// TwinCAT 3 PLC project PLC
// ProgramVersion: 3.1.4024.0
// libraries:
//   SPT Base Types, * (Beckhoff Automation LLC)
//   SPT Components, * (Beckhoff Automation LLC)
//   SPT Diagnostic, * (Beckhoff Automation LLC)
//   SPT EtherCat, * (Beckhoff Automation LLC)
//   SPT Event Logger, * (Beckhoff Automation LLC)
//   SPT Kinematics, * (Beckhoff Automation LLC)
//   SPT Motion Control, * (Beckhoff Automation LLC)
//   SPT NCI, * (Beckhoff Automation LLC)
//   SPT Utilities, * (Beckhoff Automation LLC)
//   SPT Vision, * (Beckhoff Automation LLC)
//   SPT XTS, * (Beckhoff Automation LLC)
//   Tc2_MC2_Camming, * (Beckhoff Automation GmbH)
//   Tc2_Standard, * (Beckhoff Automation GmbH)
//   Tc2_System, * (Beckhoff Automation GmbH)
//   Tc3_Module, * (Beckhoff Automation GmbH)
//   VisuDialogs, * (System)
//   Tc2_EtherCAT,newest,Beckhoff Automation GmbH
//   Tc2_Math,newest,Beckhoff Automation GmbH
//   Tc2_MC2,newest,Beckhoff Automation GmbH
//   Tc2_MC2_Drive,newest,Beckhoff Automation GmbH
//   Tc2_Utilities,newest,Beckhoff Automation GmbH
//   Tc3_EventLogger,newest,Beckhoff Automation GmbH
//   Tc3_IPCDiag,newest,Beckhoff Automation GmbH
//   Tc3_JsonXml,newest,Beckhoff Automation GmbH
//   Tc3_MC2_AdvancedHoming,newest,Beckhoff Automation GmbH
//   Tc3_PackML_V2,newest,Beckhoff Automation GmbH
// project tree:
//   / GlobalTextList.TcGTLO (not stored), PlcTask.TcTTO (not stored), Visualization Manager.TcVMO (not stored)
//   Machine/EquipmentModules/ FB_MainDrive.TcPOU, FB_Station1.TcPOU, FB_Station2.TcPOU, FB_Station3.TcPOU, FB_Station4.TcPOU, FB_Station5.TcPOU
//   Machine/MachineModule/ FB_Machine.TcPOU
//   POUs/ MAIN.TcPOU
//   VISUs/ V_Operation.TcVIS, V_Machine.TcVIS
// real-time tasks:
//   TASK PlcTask: cycle T#10ms, priority 20, ADS port 350
// motion (NC):
//   TASK NC-Task 1 SAF: cycle T#2ms, priority 4, ADS port 501
//   TASK NC-Task 1 SVB: cycle T#10ms, priority 8, ADS port 511
//   AXIS Fixed Axis (id 2)
//   AXIS Variable Axis (id 3)
//   AXIS Virtual Cammed Axis (id 4)
//   AXIS Cammed Axis (id 5)
//   AXIS Virtual Offset Master Axis 4 (id 8)
//   AXIS Offset Axis (id 7)
//   AXIS Virtual Cammed Master Axis (id 9)
//   AXIS Cammed Offset Axis (id 10)
//   AXIS Virtual Offset Master Axis 5 (id 6)
//   AXIS Machine Virtual Axis (id 1)
// variable links:
//   PLC/PLC Instance <-> NC-Task 1 SAF/Axes/Cammed Axis
//     PlcTask Inputs/MAIN.Machine.Station3.CammedAxis.BasicSlaveAxis._Axis.NcToPlc <-> Outputs/ToPlc
//     PlcTask Outputs/MAIN.Machine.Station3.CammedAxis.BasicSlaveAxis._Axis.PlcToNc <-> Inputs/FromPlc
//   PLC/PLC Instance <-> NC-Task 1 SAF/Axes/Cammed Offset Axis
//     PlcTask Inputs/MAIN.Machine.Station5.CammedOffsetAxis.BasicSlaveAxis._Axis.NcToPlc <-> Outputs/ToPlc
//     PlcTask Outputs/MAIN.Machine.Station5.CammedOffsetAxis.BasicSlaveAxis._Axis.PlcToNc <-> Inputs/FromPlc
//   PLC/PLC Instance <-> NC-Task 1 SAF/Axes/Fixed Axis
//     PlcTask Inputs/MAIN.Machine.Station1.FixedAxis.BasicSlaveAxis._Axis.NcToPlc <-> Outputs/ToPlc
//     PlcTask Outputs/MAIN.Machine.Station1.FixedAxis.BasicSlaveAxis._Axis.PlcToNc <-> Inputs/FromPlc
//   PLC/PLC Instance <-> NC-Task 1 SAF/Axes/Machine Virtual Axis
//     PlcTask Inputs/MAIN.Machine.MainDrive.MachineVirtualAxis.BasicAxis._Axis.NcToPlc <-> Outputs/ToPlc
//     PlcTask Outputs/MAIN.Machine.MainDrive.MachineVirtualAxis.BasicAxis._Axis.PlcToNc <-> Inputs/FromPlc
//   PLC/PLC Instance <-> NC-Task 1 SAF/Axes/Offset Axis
//     PlcTask Inputs/MAIN.Machine.Station4.OffsetAxis.BasicSlaveAxis._Axis.NcToPlc <-> Outputs/ToPlc
//     PlcTask Outputs/MAIN.Machine.Station4.OffsetAxis.BasicSlaveAxis._Axis.PlcToNc <-> Inputs/FromPlc
//   PLC/PLC Instance <-> NC-Task 1 SAF/Axes/Variable Axis
//     PlcTask Inputs/MAIN.Machine.Station2.VariableAxis.BasicSlaveAxis._Axis.NcToPlc <-> Outputs/ToPlc
//     PlcTask Outputs/MAIN.Machine.Station2.VariableAxis.BasicSlaveAxis._Axis.PlcToNc <-> Inputs/FromPlc
//   PLC/PLC Instance <-> NC-Task 1 SAF/Axes/Virtual Cammed Axis
//     PlcTask Inputs/MAIN.Machine.Station3.VirtualCammedAxis.CamSlaveAxis._Axis.NcToPlc <-> Outputs/ToPlc
//     PlcTask Outputs/MAIN.Machine.Station3.VirtualCammedAxis.CamSlaveAxis._Axis.PlcToNc <-> Inputs/FromPlc
//   PLC/PLC Instance <-> NC-Task 1 SAF/Axes/Virtual Cammed Master Axis
//     PlcTask Inputs/MAIN.Machine.Station5.VirtualCammedMasterAxis.CamSlaveAxis._Axis.NcToPlc <-> Outputs/ToPlc
//     PlcTask Outputs/MAIN.Machine.Station5.VirtualCammedMasterAxis.CamSlaveAxis._Axis.PlcToNc <-> Inputs/FromPlc
//   PLC/PLC Instance <-> NC-Task 1 SAF/Axes/Virtual Offset Master Axis 4
//     PlcTask Inputs/MAIN.Machine.Station4.VirtualOffsetMasterAxis.BasicAxis._Axis.NcToPlc <-> Outputs/ToPlc
//     PlcTask Outputs/MAIN.Machine.Station4.VirtualOffsetMasterAxis.BasicAxis._Axis.PlcToNc <-> Inputs/FromPlc
//   PLC/PLC Instance <-> NC-Task 1 SAF/Axes/Virtual Offset Master Axis 5
//     PlcTask Inputs/MAIN.Machine.Station5.VirtualOffsetMasterAxis.BasicAxis._Axis.NcToPlc <-> Outputs/ToPlc
//     PlcTask Outputs/MAIN.Machine.Station5.VirtualOffsetMasterAxis.BasicAxis._Axis.PlcToNc <-> Inputs/FromPlc

// ---- Machine/EquipmentModules/FB_MainDrive.TcPOU
FUNCTION_BLOCK FB_MainDrive EXTENDS FB_PackML_BaseModule
VAR
	MachineVirtualAxis : FB_Component_BasicAxis := (Name := 'Machine Virtual Axis');
	_StartCommand	   : BOOL;
END_VAR

(*
	Components:
		MachineVirtualAxis - will serve as the Master axis for all station axes to follow.
	
	Methods:
		Execute - Provides a reversing sequece from 0 to 1080 for the MachineVirtualAxis
			1080 is used because it is evenly divisible by 360, which is used as the rollover for the Cam table master position.
		Initialize - Sets MachineVirtualAxis velocity to 100, can be later adjusted by Visu

*)

METHOD PROTECTED Aborting
//Mode is ignored
CASE SequenceState OF
	0:
		NoStateTasksToComplete := FALSE;
		SequenceState		   := SequenceState + 10;

	10: (* Stop Axis *)
		MachineVirtualAxis.Override := 100;
		IF MachineVirtualAxis.Stop() THEN
			SequenceState := SequenceState + 10;
		END_IF

	20:
		IF MachineVirtualAxis.Stopped THEN
			SequenceState := SequenceState + 10;
		END_IF

	30: (* Disable Axis *)
		IF MachineVirtualAxis.Disable() THEN
			SequenceState := SequenceState + 10;
		END_IF

	40:
		IF NOT MachineVirtualAxis.Enabled THEN
			SequenceState := SequenceState + 10;
		END_IF

	50:
		StateTasksComplete := TRUE;
END_CASE

SUPER^.Aborting();
END_METHOD

PROPERTY AxisRef : REFERENCE TO AXIS_REF
GET
AxisRef REF= MachineVirtualAxis.Axis;
END_GET
END_PROPERTY

METHOD PROTECTED Completing
CASE _CurrentMode OF
	ePMLUnitMode_Production:
		CASE SequenceState OF
			0:
				NoStateTasksToComplete := FALSE;
				SequenceState		   := SequenceState + 10;

			10:
				IF MachineVirtualAxis.Stop() THEN
					SequenceState := SequenceState + 10;
				END_IF

			20:
				IF MachineVirtualAxis.Stopped THEN
					SequenceState := SequenceState + 10;
				END_IF

			30:
				StateTasksComplete := TRUE;
		END_CASE
END_CASE

SUPER^.Completing();
END_METHOD

METHOD PUBLIC CyclicLogic
IF NOT InitComplete THEN
	_InitComplete := Initialize();
	RETURN;
END_IF

SUPER^.CyclicLogic();
END_METHOD

METHOD PROTECTED Execute
VAR
END_VAR
CASE _CurrentMode OF
	ePMLUnitMode_Production:
		CASE SequenceState OF
			0: //Wait for command from Machine Module
				IF _StartCommand THEN
					_StartCommand := FALSE;
					SequenceState := SequenceState + 10;
				END_IF

			10: //Steps 10 - 40 provide a reversing sequence for the MachineVirtualAxis
				IF MachineVirtualAxis.MoveAbsolute(1_080, 0) THEN
					SequenceState := SequenceState + 10;
				END_IF

			20:
				IF NOT MachineVirtualAxis.Busy THEN
					IF NOT MachineVirtualAxis.Error THEN
						SequenceState := SequenceState + 10;
					END_IF
				END_IF

			30:
				IF MachineVirtualAxis.MoveAbsolute(0, 0) THEN
					SequenceState := SequenceState + 10;
				END_IF

			40:
				IF NOT MachineVirtualAxis.Busy THEN
					IF NOT MachineVirtualAxis.Error THEN
						SequenceState := 10;
					END_IF
				END_IF
		END_CASE
END_CASE
END_METHOD

METHOD PROTECTED Initialize : BOOL
Initialize := FALSE;
CASE DescendantSequenceState OF
	0:
		RegisterComponent(Component := MachineVirtualAxis);
		MachineVirtualAxis.Velocity := 100.0;
		DescendantSequenceState		:= DescendantSequenceState + 10;

	10:
		IF SUPER^.Initialize() THEN
			DescendantSequenceState := DescendantSequenceState + 10;
		END_IF

	20:
		Initialize := TRUE;
END_CASE
END_METHOD

PROPERTY StartCommand : BOOL
SET
_StartCommand := StartCommand;
END_SET
END_PROPERTY

METHOD PROTECTED Starting
CASE _CommandedMode OF
	ePMLProtUnitMode_Production:
		CASE SequenceState OF
			0:
				NoStateTasksToComplete := FALSE;
				SequenceState		   := SequenceState + 10;

			10:
				IF MachineVirtualAxis.Enable() THEN
					SequenceState := SequenceState + 10;
				END_IF

			20:
				IF MachineVirtualAxis.Enabled THEN
					SequenceState := SequenceState + 10;
				END_IF

			30:
				IF MachineVirtualAxis.MoveAbsolute(0, 0) THEN
					SequenceState := SequenceState + 10;
				END_IF

			40:
				IF NOT MachineVirtualAxis.Busy THEN
					IF NOT machinevirtualaxis.Error THEN
						SequenceState := SequenceState + 10;
					END_IF
				END_IF

			50:
				StateTasksComplete := TRUE;
		END_CASE
END_CASE

SUPER^.Starting();
END_METHOD

METHOD PROTECTED Stopping
CASE _CurrentMode OF
	ePMLUnitMode_Production:
		CASE SequenceState OF
			0:
				NoStateTasksToComplete := FALSE;
				SequenceState		   := SequenceState + 10;

			10:
				IF MachineVirtualAxis.Stop() THEN
					SequenceState := SequenceState + 10;
				END_IF

			20:
				IF MachineVirtualAxis.Stopped THEN
					SequenceState := SequenceState + 10;
				END_IF

			30:
				StateTasksComplete := TRUE;
		END_CASE
END_CASE

SUPER^.Stopping();
END_METHOD

END_FUNCTION_BLOCK

// ---- Machine/EquipmentModules/FB_Station1.TcPOU
FUNCTION_BLOCK FB_Station1 EXTENDS FB_PackML_BaseModule
VAR
	FixedAxis  : FB_Component_BasicSlaveAxis := (Name := 'Station 1 Fixed Axis');
	_MasterRef : REFERENCE TO AXIS_REF;
END_VAR

(*
	Component for FixedAxis that follows the MachineVirtualAxis at a fixed Gear Ratio

	Methods:
		Initialize - 
			Set the Component (FixedAxis) Master1 axis Ref to the Property backer variable for _MasterAxisRef after the component is initialized
			
		Starting - 
			Set the Gear Ratio
			Couples axis
			
*)

METHOD PROTECTED Aborting
//Mode is ignored
CASE SequenceState OF
	0:
		NoStateTasksToComplete := FALSE;
		SequenceState		   := SequenceState + 10;

	10: (* Stop Axis *)

		//Setting Override to 100 will ensure velocity calculations are not limited
		FixedAxis.Override := 100;
		IF FixedAxis.Stop() THEN //This will also GearOut by default
			SequenceState := SequenceState + 10;
		END_IF

	20:
		IF FixedAxis.Stopped THEN
			SequenceState := SequenceState + 10;
		END_IF

	30: (* Disable Axis *)
		IF FixedAxis.Disable() THEN
			SequenceState := SequenceState + 10;
		END_IF

	40:
		IF NOT FixedAxis.Enabled THEN
			SequenceState := SequenceState + 10;
		END_IF

	50:
		StateTasksComplete := TRUE;
END_CASE

SUPER^.Aborting();
END_METHOD

METHOD PROTECTED Completing
CASE _CurrentMode OF
	ePMLUnitMode_Production:
		CASE SequenceState OF
			0:
				NoStateTasksToComplete := FALSE;
				SequenceState		   := SequenceState + 10;

			10:
				IF FixedAxis.Stop() THEN //This will also GearOut
					SequenceState := SequenceState + 10;
				END_IF

			20:
				IF FixedAxis.Stopped THEN
					SequenceState := SequenceState + 10;
				END_IF

			30:
				StateTasksComplete := TRUE;
		END_CASE
END_CASE

SUPER^.Completing();
END_METHOD

METHOD PUBLIC CyclicLogic
IF NOT InitComplete THEN
	_InitComplete := Initialize();
	RETURN;
END_IF

SUPER^.CyclicLogic();
END_METHOD

METHOD PROTECTED Initialize : BOOL;
Initialize := FALSE;
CASE DescendantSequenceState OF
	0:
		RegisterComponent(FixedAxis);
		DescendantSequenceState := DescendantSequenceState + 10;

	10:
		IF SUPER^.Initialize() THEN
			//Setting the Reference of the FB_Component_BasicSlaveAxis must be done after the component has been initialized
			FixedAxis.Master1		REF= _MasterRef;
			DescendantSequenceState := DescendantSequenceState + 10;
		END_IF

	20:
		Initialize := TRUE;
END_CASE
END_METHOD

PROPERTY MasterAxisRef : REFERENCE TO AXIS_REF
SET
_MasterRef REF= MasterAxisRef;
END_SET
END_PROPERTY

METHOD PROTECTED Starting
CASE _CommandedMode OF
	ePMLProtUnitMode_Production:
		CASE SequenceState OF
			0:
				NoStateTasksToComplete := FALSE;
				SequenceState		   := SequenceState + 10;

			10: (* Enable Axis *)
				IF FixedAxis.Enable() THEN
					SequenceState := SequenceState + 10;
				END_IF

			20:
				IF FixedAxis.Enabled THEN
					SequenceState := SequenceState + 10;
				END_IF

			30:
				IF FixedAxis.MoveAbsolute(0, 0) THEN
					SequenceState := SequenceState + 10;
				END_IF

			40:
				IF NOT FixedAxis.Busy THEN
					IF NOT FixedAxis.Error THEN
						SequenceState := SequenceState + 10;
					END_IF
				END_IF

			50: (* Verify the Master axis is ready *)
				IF FixedAxis.Master1.Status.Operational THEN
					IF FixedAxis.Master1.NcToPlc.ActPos = 0.0 THEN
						SequenceState := SequenceState + 10;
					END_IF
				END_IF

			60: (* Couple to Master axis *)
				FixedAxis.RatioMaster1 := 0.5;
				IF FixedAxis.GearIn() THEN
					SequenceState := SequenceState + 10;
				END_IF

			70:
				IF FixedAxis.InGear THEN
					SequenceState := SequenceState + 10;
				END_IF

			80:
				StateTasksComplete := TRUE;
		END_CASE
END_CASE

SUPER^.Starting();
END_METHOD

METHOD PROTECTED Stopping
CASE _CurrentMode OF
	ePMLUnitMode_Production:
		CASE SequenceState OF
			0:
				NoStateTasksToComplete := FALSE;
				SequenceState		   := SequenceState + 10;

			10:
				IF FixedAxis.Stop() THEN //This will also GearOut by default
					SequenceState := SequenceState + 10;
				END_IF

			20:
				IF FixedAxis.Stopped THEN
					SequenceState := SequenceState + 10;
				END_IF

			30:
				StateTasksComplete := TRUE;
		END_CASE
END_CASE

SUPER^.Stopping();
END_METHOD

END_FUNCTION_BLOCK

// ---- Machine/EquipmentModules/FB_Station2.TcPOU
FUNCTION_BLOCK FB_Station2 EXTENDS FB_PackML_BaseModule
VAR
	VariableAxis	  : FB_Component_BasicSlaveAxis := (Name := 'Station 2 Variable Axis');
	_MasterRef		  : REFERENCE TO AXIS_REF;
	variableGearRatio : LREAL := 1.0;
	sync			  : BOOL  := TRUE;
END_VAR

(*
	Component for VariableAxis that follows the MachineVirtualAxis at a Variable Gear Ratio

	Methods:
		CyclicLogic:
			Monitors the Check Box on the Visu and changes the Gear Ratio as selected
	
		Initialize - 
			Set the Component (VariableAxis) Master1 axis Ref to the Property backer variable for _MasterAxisRef after the component is initialized

	
		Starting - 
			Set the Gear Ratio to variableGearRatio which has a default of 1.0 and can be changed from the Visu
			Couples axis

*)

METHOD PROTECTED Aborting
//Mode is ignored
CASE SequenceState OF
	0:
		NoStateTasksToComplete := FALSE;
		SequenceState		   := SequenceState + 10;

	10: (* Stop Axis *)

		//Setting Override to 100 will ensure velocity calculations are not limited
		VariableAxis.Override := 100;
		IF VariableAxis.Stop() THEN //This will also GearOut
			SequenceState := SequenceState + 10;
		END_IF

	20:
		IF VariableAxis.Stopped THEN
			SequenceState := SequenceState + 10;
		END_IF

	30: (* Disable Axis *)
		IF VariableAxis.Disable() THEN
			SequenceState := SequenceState + 10;
		END_IF

	40:
		IF NOT VariableAxis.Enabled THEN
			SequenceState := SequenceState + 10;
		END_IF

	50:
		StateTasksComplete := TRUE;
END_CASE

SUPER^.Aborting();
END_METHOD

METHOD PROTECTED Completing
CASE _CurrentMode OF
	ePMLUnitMode_Production:
		CASE SequenceState OF
			0:
				NoStateTasksToComplete := FALSE;
				SequenceState		   := SequenceState + 10;

			10:
				IF VariableAxis.Stop() THEN //This will also GearOut
					SequenceState := SequenceState + 10;
				END_IF

			20:
				IF VariableAxis.Stopped THEN
					SequenceState := SequenceState + 10;
				END_IF

			30:
				StateTasksComplete := TRUE;
		END_CASE
END_CASE

SUPER^.Completing();
END_METHOD

METHOD PUBLIC CyclicLogic
IF NOT InitComplete THEN
	_InitComplete := Initialize();
	RETURN;
END_IF

//Change at Master 0 Position? Selectable in Visu
IF sync THEN
	IF _MasterRef.NcToPlc.ActPos = 0.0 THEN
		VariableAxis.RatioMaster1 := variableGearRatio;
	END_IF
ELSE
	VariableAxis.RatioMaster1 := variableGearRatio;
END_IF

//
SUPER^.CyclicLogic();
END_METHOD

METHOD PROTECTED Initialize : BOOL;
Initialize := FALSE;
CASE DescendantSequenceState OF
	0:
		RegisterComponent(VariableAxis);
		DescendantSequenceState := DescendantSequenceState + 10;

	10:
		IF SUPER^.Initialize() THEN
			//Setting the Reference of the FB_Component_BasicSlaveAxis must be done after the component has been initialized
			VariableAxis.Master1	REF= _MasterRef;
			DescendantSequenceState := DescendantSequenceState + 10;
		END_IF

	20:
		Initialize := TRUE;
END_CASE
END_METHOD

PROPERTY MasterAxisRef : REFERENCE TO AXIS_REF
SET
_MasterRef REF= MasterAxisRef;
END_SET
END_PROPERTY

METHOD PROTECTED Starting
CASE _CommandedMode OF
	ePMLProtUnitMode_Production:
		CASE SequenceState OF
			0:
				NoStateTasksToComplete := FALSE;
				SequenceState		   := SequenceState + 10;

			10: (* Enable Axis *)
				IF VariableAxis.Enable() THEN
					SequenceState := SequenceState + 10;
				END_IF

			20:
				IF VariableAxis.Enabled THEN
					SequenceState := SequenceState + 10;
				END_IF

			30:
				IF VariableAxis.MoveAbsolute(0, 0) THEN
					SequenceState := SequenceState + 10;
				END_IF

			40:
				IF NOT VariableAxis.Busy THEN
					IF NOT VariableAxis.Error THEN
						SequenceState := SequenceState + 10;
					END_IF
				END_IF

			50: (* Verify the Master axis is ready *)
				IF VariableAxis.Master1.Status.Operational THEN
					IF VariableAxis.Master1.NcToPlc.ActPos = 0.0 THEN
						SequenceState := SequenceState + 10;
					END_IF
				END_IF

			60: (* Couple to Master axis *)
				VariableAxis.RatioMaster1 := variableGearRatio;
				IF VariableAxis.GearIn() THEN
					SequenceState := SequenceState + 10;
				END_IF

			70:
				IF VariableAxis.InGear THEN
					SequenceState := SequenceState + 10;
				END_IF

			80:
				StateTasksComplete := TRUE;
		END_CASE
END_CASE

SUPER^.Starting();
END_METHOD

METHOD PROTECTED Stopping
CASE _CurrentMode OF
	ePMLUnitMode_Production:
		CASE SequenceState OF
			0:
				NoStateTasksToComplete := FALSE;
				SequenceState		   := SequenceState + 10;

			10:
				IF VariableAxis.Stop() THEN //This will also GearOut by default
					SequenceState := SequenceState + 10;
				END_IF

			20:
				IF VariableAxis.Stopped THEN
					SequenceState := SequenceState + 10;
				END_IF

			30:
				StateTasksComplete := TRUE;
		END_CASE
END_CASE

SUPER^.Stopping();
END_METHOD

END_FUNCTION_BLOCK

// ---- Machine/EquipmentModules/FB_Station3.TcPOU
FUNCTION_BLOCK FB_Station3 EXTENDS FB_PackML_BaseModule
VAR
	VirtualCammedAxis : FB_Component_CamSlaveAxis	:= (Name := 'Station 3 Virtual Cammed Axis');
	CammedAxis		  : FB_Component_BasicSlaveAxis := (Name := 'Station 3 Cammed Axis');
	_MasterRef		  : REFERENCE TO AXIS_REF;
	CamParameters	  : ST_CamParameters;
END_VAR

(*
	Design Considerations:
		Why use a Virtual Axis?
			Software/Virtual axes can be easily managed from within TwinCAT PLC and NC. 
			Notably the encoder value can be changed without physical movement and with no impact to real hardware.
			Therefore, it is possible to set position on a virtual axis to a specific value without physical movement an with no impact to the coupled axis.

			When using a Virtual axis for a Cam table, the real axis can be decoupled, 
			then the virtual cam table slave can be adjusted as needed, and then the real axis can couple to the virtual axis.
						
	
	Components:
		VirtualCammedAxis - follows the cam table with the MachineVirtualAxis as the master axis of the table.
			The Cam table is a move from 0 - 100
		CammedAxis - geared to the Virtual Cammed Axis at the default ratio of 1.

	Methods:
		Initialize - 
			Create the Cam table data and set the Component (VirtualCammedAxis) CamParameters Ref to the data after the component is initialized
			Set the Component (VirtualCammedAxis) Master axis Ref to the Property backer variable for _MasterAxisRef after the component is initialized
			Set the Component (CammedAxis) Master1 axis Ref to the Component (VirtualCammedAxis) Axis property
			
	
	
		Starting - 
			Calls StartSync method of VirtualCammedAxis to cam axis to table
			Couple Cammed Axis to VirtualCammedAxis
			
*)

METHOD PROTECTED Aborting
//Mode is ignored
CASE SequenceState OF
	0:
		NoStateTasksToComplete := FALSE;
		SequenceState		   := SequenceState + 10;

	10: (* Stop Axis *)

		//Setting Override to 100 will ensure velocity calculations are not limited
		VirtualCammedAxis.Override := 100;
		CammedAxis.Override		   := 100;
		IF VirtualCammedAxis.Stop() THEN //This will also GearOut by default
			SequenceState := SequenceState + 10;
		END_IF

	20:
		IF CammedAxis.Stop() THEN //This will also GearOut by default
			SequenceState := SequenceState + 10;
		END_IF

	30:
		IF VirtualCammedAxis.Stopped AND CammedAxis.Stopped THEN
			SequenceState := SequenceState + 10;
		END_IF

	40: (* Disable Axis *)
		IF VirtualCammedAxis.Disable() THEN
			SequenceState := SequenceState + 10;
		END_IF

	50:
		IF CammedAxis.Disable() THEN
			SequenceState := SequenceState + 10;
		END_IF

	60:
		IF NOT VirtualCammedAxis.Enabled AND NOT CammedAxis.Enabled THEN
			SequenceState := SequenceState + 10;
		END_IF

	70:
		StateTasksComplete := TRUE;
END_CASE

SUPER^.Aborting();
END_METHOD

METHOD PROTECTED Completing
CASE SequenceState OF
	0:
		NoStateTasksToComplete := FALSE;
		SequenceState		   := SequenceState + 10;

	10:
		IF VirtualCammedAxis.Stop() THEN //This will also GearOut
			SequenceState := SequenceState + 10;
		END_IF

	20:
		IF CammedAxis.Stop() THEN
			SequenceState := SequenceState + 10;
		END_IF

	30:
		IF VirtualCammedAxis.Stopped AND CammedAxis.Stopped THEN
			SequenceState := SequenceState + 10;
		END_IF

	40:
		StateTasksComplete := TRUE;
END_CASE

SUPER^.Completing();
END_METHOD

METHOD PUBLIC CyclicLogic
IF NOT InitComplete THEN
	_InitComplete := Initialize();
	RETURN;
END_IF

//
SUPER^.CyclicLogic();
END_METHOD

METHOD PROTECTED Initialize : BOOL;
Initialize := FALSE;
CASE DescendantSequenceState OF
	0:
		RegisterComponent(VirtualCammedAxis);
		RegisterComponent(CammedAxis);
		DescendantSequenceState := DescendantSequenceState + 10;

	10:
		IF SUPER^.Initialize() THEN
			//Create the Cam table data and set the Component (VirtualCammedAxis) CamParameters Ref to the data after the component is initialized
			WriteCamParameters();
			VirtualCammedAxis.CamParameters REF= CamParameters;

			//Setting the Reference of the FB_Component_CamSlaveAxis must be done after the component has been initialized
			VirtualCammedAxis.Master REF= _MasterRef;

			//Setting the Reference of the FB_Component_BasicSlaveAxis must be done after the component has been initialized
			CammedAxis.Master1 REF= VirtualCammedAxis.Axis;

			//
			DescendantSequenceState := DescendantSequenceState + 10;
		END_IF

	20:
		Initialize := TRUE;
END_CASE
END_METHOD

PROPERTY MasterAxisRef : REFERENCE TO AXIS_REF
SET
_MasterRef REF= MasterAxisRef;
END_SET
END_PROPERTY

METHOD PROTECTED Starting
CASE _CommandedMode OF
	ePMLProtUnitMode_Production:
		CASE SequenceState OF
			0:
				NoStateTasksToComplete := FALSE;
				SequenceState		   := SequenceState + 10;

			10: (* Enable Axis *)
				IF VirtualCammedAxis.Enable() THEN
					SequenceState := SequenceState + 10;
				END_IF

			20:
				IF VirtualCammedAxis.Enabled THEN
					SequenceState := SequenceState + 10;
				END_IF

			30:
				IF VirtualCammedAxis.MoveAbsolute(0, 0) THEN
					SequenceState := SequenceState + 10;
				END_IF

			40:
				IF NOT VirtualCammedAxis.Busy THEN
					IF NOT VirtualCammedAxis.Error THEN
						SequenceState := SequenceState + 10;
					END_IF
				END_IF

			50: (* Enable Axis *)
				IF CammedAxis.Enable() THEN
					SequenceState := SequenceState + 10;
				END_IF

			60:
				IF CammedAxis.Enabled THEN
					SequenceState := SequenceState + 10;
				END_IF

			70:
				IF CammedAxis.MoveAbsolute(0, 0) THEN
					SequenceState := SequenceState + 10;
				END_IF

			80:
				IF NOT CammedAxis.Busy THEN
					IF NOT CammedAxis.Error THEN
						SequenceState := SequenceState + 10;
					END_IF
				END_IF

			90: (* Verify the Master axis is ready *)
				IF VirtualCammedAxis.Master.Status.Operational THEN
					IF VirtualCammedAxis.Master.NcToPlc.ActPos = 0.0 THEN
						SequenceState := SequenceState + 10;
					END_IF
				END_IF

			100: (* Couple to Cam table with Master axis*)
				IF VirtualCammedAxis.StartSync() THEN
					SequenceState := SequenceState + 10;
				END_IF

			110:
				IF VirtualCammedAxis.InSync THEN
					SequenceState := SequenceState + 10;
				END_IF

			120: (* Verify the Master axis is ready *)
				IF CammedAxis.Master1.Status.Operational THEN
					//A small tolerance of position is used becaused the Axis moves by a small amount when cammed in 
					IF CammedAxis.Master1.NcToPlc.ActPos <= 0.01 AND CammedAxis.Master1.NcToPlc.ActPos >= -0.01 THEN
						SequenceState := SequenceState + 10;
					END_IF
				END_IF

			130: (*Couple to Master Axis*)
				IF CammedAxis.GearIn() THEN
					SequenceState := SequenceState + 10;
				END_IF

			140:
				IF CammedAxis.InGear THEN
					SequenceState := SequenceState + 10;
				END_IF

			150:
				StateTasksComplete := TRUE;
		END_CASE
END_CASE

SUPER^.Starting();
END_METHOD

METHOD PROTECTED Stopping
CASE SequenceState OF
	0:
		NoStateTasksToComplete := FALSE;
		SequenceState		   := SequenceState + 10;

	10:
		IF VirtualCammedAxis.Stop() THEN //This will also GearOut by default
			SequenceState := SequenceState + 10;
		END_IF

	20:
		IF CammedAxis.Stop() THEN //This will also GearOut by default
			SequenceState := SequenceState + 10;
		END_IF

	30:
		IF VirtualCammedAxis.Stopped AND CammedAxis.Stopped THEN
			SequenceState := SequenceState + 10;
		END_IF

	40:
		StateTasksComplete := TRUE;
END_CASE

SUPER^.Stopping();
END_METHOD

METHOD WriteCamParameters
CamParameters.CamTableId := VirtualCammedAxis.Axis.NcToPlc.AxisId;

//Table 1
CamParameters.CamTable[1].NumberOfPoints			  := 3;
CamParameters.CamTable[1].Points[1].PointIndex		  := 1;
CamParameters.CamTable[1].Points[1].FunctionType	  := MC_MotionFunctionType.MOTIONFUNCTYPE_POLYNOM5;
CamParameters.CamTable[1].Points[1].PointType		  := MC_MotionPointType.MOTIONPOINTTYPE_REST;
CamParameters.CamTable[1].Points[1].RelIndexNextPoint := 1;
CamParameters.CamTable[1].Points[1].MasterPos		  := 0.0;
CamParameters.CamTable[1].Points[1].SlavePos		  := 0.0;
CamParameters.CamTable[1].Points[2].PointIndex		  := 2;
CamParameters.CamTable[1].Points[2].FunctionType	  := MC_MotionFunctionType.MOTIONFUNCTYPE_POLYNOM5;
CamParameters.CamTable[1].Points[2].PointType		  := MC_MotionPointType.MOTIONPOINTTYPE_TURN;
CamParameters.CamTable[1].Points[2].RelIndexNextPoint := 1;
CamParameters.CamTable[1].Points[2].MasterPos		  := 180.0;
CamParameters.CamTable[1].Points[2].SlavePos		  := 100.0;
CamParameters.CamTable[1].Points[3].PointIndex		  := 3;
CamParameters.CamTable[1].Points[3].FunctionType	  := MC_MotionFunctionType.MOTIONFUNCTYPE_POLYNOM5;
CamParameters.CamTable[1].Points[3].PointType		  := MC_MotionPointType.MOTIONPOINTTYPE_REST;
CamParameters.CamTable[1].Points[3].RelIndexNextPoint := 0;
CamParameters.CamTable[1].Points[3].MasterPos		  := 360.0;
CamParameters.CamTable[1].Points[3].SlavePos		  := 0.0;
CamParameters.CamTable[1].NumberOfPoints			  := 3;
END_METHOD

END_FUNCTION_BLOCK

// ---- Machine/EquipmentModules/FB_Station4.TcPOU
FUNCTION_BLOCK FB_Station4 EXTENDS FB_PackML_BaseModule
VAR
	VirtualOffsetMasterAxis : FB_Component_BasicAxis	  := (Name := 'Station 4 Virtual Offset Master Axis');
	OffsetAxis				: FB_Component_BasicSlaveAxis := (Name := 'Station 4 Offset Axis');
	_MasterRef				: REFERENCE TO AXIS_REF;
	V_OffsetFWD				: BOOL;
	V_OffsetREV				: BOOL;
END_VAR

(*
	Components:
		VirtualOffsetMasterAxis - Local virtual axis used to apply an offset to the real axis position
		OffsetAxis - geared to the MachineVirtualAxis and the VirtualOffsetMasterAxis, and will follow commands from both.

	Methods:
		CyclicLogic - 
			Monitors the HMI variables to move the VirtualOffsetMasterAxis +/- 100

		Initialize - 
			Set the Component Master1 axis Ref to the Property backer variable for _MasterAxisRef after the component is initialized
			Set the Component Master2 axis Ref to the VirtualOffsetMasterAxis.Axis after the component is initialized
	
		Starting - 
			Couples the OffsetAxis to both master axes		

*)

METHOD PROTECTED Aborting
//Mode is ignored
CASE SequenceState OF
	0:
		NoStateTasksToComplete := FALSE;
		SequenceState		   := SequenceState + 10;

	10: //Setting Override to 100 will ensure velocity calculations are not limited
		VirtualOffsetMasterAxis.Override := 100;
		OffsetAxis.Override				 := 100;
		IF VirtualOffsetMasterAxis.Stop() THEN //This will also GearOut by default
			SequenceState := SequenceState + 10;
		END_IF

	20:
		IF OffsetAxis.Stop() THEN //This will also GearOut by default
			SequenceState := SequenceState + 10;
		END_IF

	30:
		IF VirtualOffsetMasterAxis.Stopped AND OffsetAxis.Stopped THEN
			SequenceState := SequenceState + 10;
		END_IF

	40: (* Disable Axis *)
		IF VirtualOffsetMasterAxis.Disable() THEN
			SequenceState := SequenceState + 10;
		END_IF

	50: (* Disable Axis *)
		IF OffsetAxis.Disable() THEN
			SequenceState := SequenceState + 10;
		END_IF

	60:
		IF NOT VirtualOffsetMasterAxis.Enabled AND NOT OffsetAxis.Enabled THEN
			SequenceState := SequenceState + 10;
		END_IF

	70:
		StateTasksComplete := TRUE;
END_CASE

SUPER^.Aborting();
END_METHOD

METHOD PROTECTED Completing
CASE SequenceState OF
	0:
		NoStateTasksToComplete := FALSE;
		SequenceState		   := SequenceState + 10;

	10:
		IF VirtualOffsetMasterAxis.Stop() THEN //This will also GearOut
			SequenceState := SequenceState + 10;
		END_IF

	20:
		IF OffsetAxis.Stop() THEN //This will also GearOut
			SequenceState := SequenceState + 10;
		END_IF

	30:
		IF VirtualOffsetMasterAxis.Stopped AND OffsetAxis.Stopped THEN
			SequenceState := SequenceState + 10;
		END_IF

	40:
		StateTasksComplete := TRUE;
END_CASE

SUPER^.Completing();
END_METHOD

METHOD PUBLIC CyclicLogic
IF NOT InitComplete THEN
	_InitComplete := Initialize();
	RETURN;
END_IF

//Move commands from Visu
IF V_OffsetFWD THEN
	VirtualOffsetMasterAxis.MoveRelative(100, 0);
END_IF

IF V_OffsetREV THEN
	VirtualOffsetMasterAxis.MoveRelative(-100, 0);
END_IF

//
SUPER^.CyclicLogic();
END_METHOD

METHOD PROTECTED Initialize : BOOL;
Initialize := FALSE;
CASE DescendantSequenceState OF
	0:
		RegisterComponent(VirtualOffsetMasterAxis);
		RegisterComponent(OffsetAxis);
		DescendantSequenceState := DescendantSequenceState + 10;

	10:
		IF SUPER^.Initialize() THEN
			//Setting the Reference of the FB_Component_BasicSlaveAxis must be done after the component has been initialized
			OffsetAxis.Master1		REF= _MasterRef;
			OffsetAxis.Master2		REF= VirtualOffsetMasterAxis.Axis;
			DescendantSequenceState := DescendantSequenceState + 10;
		END_IF

	20:
		Initialize := TRUE;
END_CASE
END_METHOD

PROPERTY MasterAxisRef : REFERENCE TO AXIS_REF
SET
_MasterRef REF= MasterAxisRef;
END_SET
END_PROPERTY

METHOD PROTECTED Starting
CASE _CommandedMode OF
	ePMLProtUnitMode_Production:
		CASE SequenceState OF
			0:
				NoStateTasksToComplete := FALSE;
				SequenceState		   := SequenceState + 10;

			10: (* Enable Axis *)
				IF VirtualOffsetMasterAxis.Enable() THEN
					SequenceState := SequenceState + 10;
				END_IF

			20:
				IF VirtualOffsetMasterAxis.Enabled THEN
					SequenceState := SequenceState + 10;
				END_IF

			30:
				IF VirtualOffsetMasterAxis.MoveAbsolute(0, 0) THEN
					SequenceState := SequenceState + 10;
				END_IF

			40:
				IF NOT VirtualOffsetMasterAxis.Busy THEN
					IF NOT VirtualOffsetMasterAxis.Error THEN
						SequenceState := SequenceState + 10;
					END_IF
				END_IF

			50: (* Enable Axis *)
				IF OffsetAxis.Enable() THEN
					SequenceState := SequenceState + 10;
				END_IF

			60:
				IF OffsetAxis.Enabled THEN
					SequenceState := SequenceState + 10;
				END_IF

			70:
				IF OffsetAxis.MoveAbsolute(0, 0) THEN
					SequenceState := SequenceState + 10;
				END_IF

			80:
				IF NOT OffsetAxis.Busy THEN
					IF NOT OffsetAxis.Error THEN
						SequenceState := SequenceState + 10;
					END_IF
				END_IF

			90: (* Verify the Master axis is ready *)
				IF OffsetAxis.Master1.Status.Operational THEN
					IF (OffsetAxis.Master1.NcToPlc.ActPos = 0.0) THEN
						SequenceState := SequenceState + 10;
					END_IF
				END_IF

			100: (* Couple to both Master axes *)
				IF OffsetAxis.GearIn() THEN
					SequenceState := SequenceState + 10;
				END_IF

			110:
				IF OffsetAxis.InGear THEN
					SequenceState := SequenceState + 10;
				END_IF

			120:
				StateTasksComplete := TRUE;
		END_CASE
END_CASE

SUPER^.Starting();
END_METHOD

METHOD PROTECTED Stopping
CASE SequenceState OF
	0:
		NoStateTasksToComplete := FALSE;
		SequenceState		   := SequenceState + 10;

	10:
		IF VirtualOffsetMasterAxis.Stop() THEN //This will also GearOut by default
			SequenceState := SequenceState + 10;
		END_IF

	20:
		IF OffsetAxis.Stop() THEN //This will also GearOut by default
			SequenceState := SequenceState + 10;
		END_IF

	30:
		IF VirtualOffsetMasterAxis.Stopped AND OffsetAxis.Stopped THEN
			SequenceState := SequenceState + 10;
		END_IF

	40:
		StateTasksComplete := TRUE;
END_CASE

SUPER^.Stopping();
END_METHOD

END_FUNCTION_BLOCK

// ---- Machine/EquipmentModules/FB_Station5.TcPOU
FUNCTION_BLOCK FB_Station5 EXTENDS FB_PackML_BaseModule
VAR
	VirtualOffsetMasterAxis : FB_Component_BasicAxis	  := (Name := 'Station 5 Virtual Offset Master Axis');
	VirtualCammedMasterAxis : FB_Component_CamSlaveAxis	  := (Name := 'Station 5 Virtual Cam Axis');
	CammedOffsetAxis		: FB_Component_BasicSlaveAxis := (Name := 'Station 5 Cammed Offset Axis');
	_MasterRef				: REFERENCE TO AXIS_REF;
	CamParameters			: ST_CamParameters;
	V_OffsetFWD				: BOOL;
	V_OffsetREV				: BOOL;
END_VAR

(*
	Design Considerations:
		Why use a Virtual Axis?
			Software/Virtual axes can be easily managed from within TwinCAT PLC and NC. 
			Notably the encoder value can be changed without physical movement and with no impact to real hardware.
			Therefore, it is possible to set position on a virtual axis to a specific value without physical movement an with no impact to the coupled axis.

			When using a Virtual axis for a Cam table, the real axis can be decoupled, 
			then the virtual cam table slave can be adjusted as needed, and then the real axis can couple to the virtual axis.
						
	
	Components:
		VirtualOffsetMasterAxis - Local virtual axis used to apply an offset to the real axis position
		VirtualCammedMasterAxis - follows the cam table with the MachineVirtualAxis as the master axis of the table.
			The Cam table is a move from 0 - 100
		CammedOffsetAxis - geared to the VirtualCammedMasterAxis and the VirtualCammedMasterAxis, and will follow commands from both.

	Methods:
		CyclicLogic - 
			Monitors the HMI variables to move the VirtualOffsetMasterAxis +/- 100
			
		Initialize - 
			Create the Cam table data and set the Component (VirtualCammedMasterAxis) CamParameters Ref to the data after the component is initialized
			Set the Component (VirtualCammedMasterAxis) Master axis Ref to the Property backer variable for _MasterAxisRef after the component is initialized
			Set the Component (CammedOffsetAxis) Master1 axis Ref to the Component (VirtualCammedMasterAxis) Axis property after the component is initialized
			Set the Component (CammedOffsetAxis) Master2 axis Ref to the Component (VirtualOffsetMasterAxis) Axis property after the component is initialized
	
	
		Starting - 
			Calls StartSync method of VirtualCammedMasterAxis to cam axis to table
			Couples the CammedOffsetAxis to both master axes		
			
*)

METHOD PROTECTED Aborting
//Mode is ignored
CASE SequenceState OF
	0:
		NoStateTasksToComplete := FALSE;
		SequenceState		   := SequenceState + 10;

	10: (* Stop Axis *)

		//Setting Override to 100 will ensure velocity calculations are not limited
		VirtualOffsetMasterAxis.Override := 100;
		VirtualCammedMasterAxis.Override := 100;
		CammedOffsetAxis.Override		 := 100;

		//
		IF VirtualOffsetMasterAxis.Stop() THEN //This will also GearOut by default
			SequenceState := SequenceState + 10;
		END_IF

	20:
		IF VirtualCammedMasterAxis.Stop() THEN //This will also GearOut by default
			SequenceState := SequenceState + 10;
		END_IF

	30:
		IF CammedOffsetAxis.Stop() THEN //This will also GearOut by default
			SequenceState := SequenceState + 10;
		END_IF

	40:
		IF VirtualOffsetMasterAxis.Stopped AND VirtualCammedMasterAxis.Stopped AND CammedOffsetAxis.Stopped THEN
			SequenceState := SequenceState + 10;
		END_IF

	50: (* Disable Axis *)
		IF VirtualOffsetMasterAxis.Disable() THEN
			SequenceState := SequenceState + 10;
		END_IF

	60: (* Disable Axis *)
		IF VirtualCammedMasterAxis.Disable() THEN
			SequenceState := SequenceState + 10;
		END_IF

	70: (* Disable Axis *)
		IF CammedOffsetAxis.Disable() THEN
			SequenceState := SequenceState + 10;
		END_IF

	80:
		IF NOT VirtualOffsetMasterAxis.Enabled AND NOT VirtualCammedMasterAxis.Enabled AND NOT CammedOffsetAxis.Enabled THEN
			SequenceState := SequenceState + 10;
		END_IF

	90:
		StateTasksComplete := TRUE;
END_CASE

SUPER^.Aborting();
END_METHOD

METHOD PROTECTED Completing
CASE SequenceState OF
	0:
		NoStateTasksToComplete := FALSE;
		SequenceState		   := SequenceState + 10;

	10:
		IF VirtualOffsetMasterAxis.Stop() THEN //This will also GearOut
			SequenceState := SequenceState + 10;
		END_IF

	20:
		IF VirtualCammedMasterAxis.Stop() THEN //This will also GearOut
			SequenceState := SequenceState + 10;
		END_IF

	30:
		IF CammedOffsetAxis.Stop() THEN //This will also GearOut
			SequenceState := SequenceState + 10;
		END_IF

	40:
		IF VirtualOffsetMasterAxis.Stopped AND VirtualCammedMasterAxis.Stopped AND CammedOffsetAxis.Stopped THEN
			SequenceState := SequenceState + 10;
		END_IF

	50:
		StateTasksComplete := TRUE;
END_CASE

SUPER^.Completing();
END_METHOD

METHOD PUBLIC CyclicLogic
IF NOT InitComplete THEN
	_InitComplete := Initialize();
	RETURN;
END_IF

//Move commands from Visu
IF V_OffsetFWD THEN
	VirtualOffsetMasterAxis.MoveRelative(100, 0);
END_IF

IF V_OffsetREV THEN
	VirtualOffsetMasterAxis.MoveRelative(-100, 0);
END_IF

//
SUPER^.CyclicLogic();
END_METHOD

METHOD PROTECTED Initialize : BOOL;
Initialize := FALSE;
CASE DescendantSequenceState OF
	0:
		RegisterComponent(VirtualOffsetMasterAxis);
		RegisterComponent(VirtualCammedMasterAxis);
		RegisterComponent(CammedOffsetAxis);
		DescendantSequenceState := DescendantSequenceState + 10;

	10:
		IF SUPER^.Initialize() THEN
			//Create the Cam table data and set the Component (VirtualCammedMasterAxis) CamParameters Ref to the data after the component is initialized
			WriteCamParameters();
			VirtualCammedMasterAxis.CamParameters REF= CamParameters;

			//Setting the Reference of the FB_Component_CamSlaveAxis must be done after the component has been initialized
			VirtualCammedMasterAxis.Master REF= _MasterRef;

			//Setting the Reference of the FB_Component_BasicSlaveAxis must be done after the component has been initialized
			CammedOffsetAxis.Master1 REF= VirtualCammedMasterAxis.Axis;
			CammedOffsetAxis.Master2 REF= VirtualOffsetMasterAxis.Axis;

			//
			DescendantSequenceState := DescendantSequenceState + 10;
		END_IF

	20:
		Initialize := TRUE;
END_CASE
END_METHOD

PROPERTY MasterAxisRef : REFERENCE TO AXIS_REF
SET
_MasterRef REF= MasterAxisRef;
END_SET
END_PROPERTY

METHOD PROTECTED Starting
CASE _CommandedMode OF
	ePMLProtUnitMode_Production:
		CASE SequenceState OF
			0:
				NoStateTasksToComplete := FALSE;
				SequenceState		   := SequenceState + 10;

			10: (* Enable Axis *)
				IF VirtualCammedMasterAxis.Enable() THEN
					SequenceState := SequenceState + 10;
				END_IF

			20:
				IF VirtualCammedMasterAxis.Enabled THEN
					SequenceState := SequenceState + 10;
				END_IF

			30:
				IF VirtualCammedMasterAxis.MoveAbsolute(0, 0) THEN
					SequenceState := SequenceState + 10;
				END_IF

			40:
				IF NOT VirtualCammedMasterAxis.Busy THEN
					IF NOT VirtualCammedMasterAxis.Error THEN
						SequenceState := SequenceState + 10;
					END_IF
				END_IF

			50: (* Enable Axis *)
				IF VirtualOffsetMasterAxis.Enable() THEN
					SequenceState := SequenceState + 10;
				END_IF

			60:
				IF VirtualOffsetMasterAxis.Enabled THEN
					SequenceState := SequenceState + 10;
				END_IF

			70:
				IF VirtualOffsetMasterAxis.MoveAbsolute(0, 0) THEN
					SequenceState := SequenceState + 10;
				END_IF

			80:
				IF NOT VirtualOffsetMasterAxis.Busy THEN
					IF NOT VirtualOffsetMasterAxis.Error THEN
						SequenceState := SequenceState + 10;
					END_IF
				END_IF

			90: (* Verify the Master axis is ready *)
				IF VirtualCammedMasterAxis.Master.Status.Operational THEN
					IF VirtualCammedMasterAxis.Master.NcToPlc.ActPos = 0.0 THEN
						SequenceState := SequenceState + 10;
					END_IF
				END_IF

			100: (* Couple to Cam table with Master axis*)
				IF VirtualCammedMasterAxis.StartSync() THEN
					SequenceState := SequenceState + 10;
				END_IF

			110:
				IF VirtualCammedMasterAxis.InSync THEN
					SequenceState := SequenceState + 10;
				END_IF

			120: (* Enable Axis *)
				IF CammedOffsetAxis.Enable() THEN
					SequenceState := SequenceState + 10;
				END_IF

			130:
				IF CammedOffsetAxis.Enabled THEN
					SequenceState := SequenceState + 10;
				END_IF

			140:
				IF CammedOffsetAxis.MoveAbsolute(0, 0) THEN
					SequenceState := SequenceState + 10;
				END_IF

			150:
				IF NOT CammedOffsetAxis.Busy THEN
					IF NOT CammedOffsetAxis.Error THEN
						SequenceState := SequenceState + 10;
					END_IF
				END_IF

			160: (* Verify the Master axis is ready *)
				IF CammedOffsetAxis.Master1.Status.Operational THEN
					//A small tolerance of position is used becaused the Axis moves by a small amount when cammed in 
					IF CammedOffsetAxis.Master1.NcToPlc.ActPos <= 0.01 AND CammedOffsetAxis.Master1.NcToPlc.ActPos >= -0.01 THEN
						SequenceState := SequenceState + 10;
					END_IF
				END_IF

			170: (* Couple to Master axis *)
				IF CammedOffsetAxis.GearIn() THEN
					SequenceState := SequenceState + 10;
				END_IF

			180:
				IF CammedOffsetAxis.InGear THEN
					SequenceState := SequenceState + 10;
				END_IF

			190:
				StateTasksComplete := TRUE;
		END_CASE
END_CASE

SUPER^.Starting();
END_METHOD

METHOD PROTECTED Stopping
CASE SequenceState OF
	0:
		NoStateTasksToComplete := FALSE;
		SequenceState		   := SequenceState + 10;

	10:
		IF VirtualOffsetMasterAxis.Stop() THEN //This will also GearOut by default
			SequenceState := SequenceState + 10;
		END_IF

	20:
		IF VirtualCammedMasterAxis.Stop() THEN //This will also GearOut by default
			SequenceState := SequenceState + 10;
		END_IF

	30:
		IF CammedOffsetAxis.Stop() THEN //This will also GearOut by default
			SequenceState := SequenceState + 10;
		END_IF

	40:
		IF VirtualOffsetMasterAxis.Stopped AND VirtualCammedMasterAxis.Stopped AND CammedOffsetAxis.Stopped THEN
			SequenceState := SequenceState + 10;
		END_IF

	50:
		StateTasksComplete := TRUE;
END_CASE

SUPER^.Stopping();
END_METHOD

METHOD WriteCamParameters
CamParameters.CamTableId := VirtualCammedMasterAxis.Axis.NcToPlc.AxisId;

//Table 1
CamParameters.CamTable[1].NumberOfPoints			  := 3;
CamParameters.CamTable[1].Points[1].PointIndex		  := 1;
CamParameters.CamTable[1].Points[1].FunctionType	  := MC_MotionFunctionType.MOTIONFUNCTYPE_POLYNOM5;
CamParameters.CamTable[1].Points[1].PointType		  := MC_MotionPointType.MOTIONPOINTTYPE_REST;
CamParameters.CamTable[1].Points[1].RelIndexNextPoint := 1;
CamParameters.CamTable[1].Points[1].MasterPos		  := 0.0;
CamParameters.CamTable[1].Points[1].SlavePos		  := 0.0;
CamParameters.CamTable[1].Points[2].PointIndex		  := 2;
CamParameters.CamTable[1].Points[2].FunctionType	  := MC_MotionFunctionType.MOTIONFUNCTYPE_POLYNOM5;
CamParameters.CamTable[1].Points[2].PointType		  := MC_MotionPointType.MOTIONPOINTTYPE_TURN;
CamParameters.CamTable[1].Points[2].RelIndexNextPoint := 1;
CamParameters.CamTable[1].Points[2].MasterPos		  := 180.0;
CamParameters.CamTable[1].Points[2].SlavePos		  := 100.0;
CamParameters.CamTable[1].Points[3].PointIndex		  := 3;
CamParameters.CamTable[1].Points[3].FunctionType	  := MC_MotionFunctionType.MOTIONFUNCTYPE_POLYNOM5;
CamParameters.CamTable[1].Points[3].PointType		  := MC_MotionPointType.MOTIONPOINTTYPE_REST;
CamParameters.CamTable[1].Points[3].RelIndexNextPoint := 0;
CamParameters.CamTable[1].Points[3].MasterPos		  := 360.0;
CamParameters.CamTable[1].Points[3].SlavePos		  := 0.0;
CamParameters.CamTable[1].NumberOfPoints			  := 3;
END_METHOD

END_FUNCTION_BLOCK

// ---- Machine/MachineModule/FB_Machine.TcPOU
{attribute 'no_explicit_call' := 'This FB is a CLASS and must be accessed using methods or properties'}
FUNCTION_BLOCK FB_Machine EXTENDS FB_PackML_BaseModule
VAR
	MainDrive : FB_MainDrive := (Name := 'Main Drive');
	Station1  : FB_Station1	 := (Name := 'Fixed Gear Ratio');
	Station2  : FB_Station2	 := (Name := 'Variable Gear Ratio');
	Station3  : FB_Station3	 := (Name := 'Cam Table');
	Station4  : FB_Station4	 := (Name := '2nd Master for Offset');
	Station5  : FB_Station5	 := (Name := '2nd Master for Offset and Cam Table');
END_VAR

(*

	Each station has a property that needs a Reference to the MachineVirtualAxis of the Main Drive.
	This is set in the Initialze method.

*)

METHOD PUBLIC CyclicLogic
IF NOT InitComplete THEN
	_InitComplete := Initialize();
	RETURN;
END_IF

SUPER^.CyclicLogic();
END_METHOD

METHOD PROTECTED Execute
CASE _CurrentMode OF
	ePMLUnitMode_Production:
		CASE SequenceState OF
			0:
				(* 
					When all EMs are in Execute the MM will change states to Execute, then the command to start the Main Drive will be given
	 				This ensures that all axes are in positin and coupled before starting the Main Drive
				*)
				MainDrive.StartCommand := TRUE;
				SequenceState		   := SequenceState + 10;

			10:
				MainDrive.StartCommand := FALSE;
		END_CASE
END_CASE
END_METHOD

METHOD PROTECTED HMIPermissions
CASE _CurrentMode OF
	E_PMLUnitMode.ePMLUnitMode_Production:
		AllowHMIControl(ThisModuleOnly := TRUE);

	E_PMLUnitMode.ePMLUnitMode_Maintenance:
		AllowHMIControl(ThisModuleOnly := FALSE);

	E_PMLUnitMode.ePMLUnitMode_Manual:
		AllowHMIControl(ThisModuleOnly := FALSE);
END_CASE
END_METHOD

METHOD PROTECTED Initialize : BOOL
Initialize := FALSE;
CASE DescendantSequenceState OF
	0:
		RegisterSubmodule(SubModule := MainDrive);
		RegisterSubmodule(SubModule := Station1);
		RegisterSubmodule(SubModule := Station2);
		RegisterSubmodule(SubModule := Station3);
		RegisterSubmodule(SubModule := Station4);
		RegisterSubmodule(SubModule := Station5);
		DescendantSequenceState := DescendantSequenceState + 10;

	10:
		//Each station has a property that needs a Reference to the MachineVirtualAxis of the Main Drive.
		Station1.MasterAxisRef	REF= MainDrive.AxisRef;
		Station2.MasterAxisRef	REF= MainDrive.AxisRef;
		Station3.MasterAxisRef	REF= MainDrive.AxisRef;
		Station4.MasterAxisRef	REF= MainDrive.AxisRef;
		Station5.MasterAxisRef	REF= MainDrive.AxisRef;
		DescendantSequenceState := DescendantSequenceState + 10;

	20:
		IF SUPER^.Initialize() THEN
			DescendantSequenceState := DescendantSequenceState + 10;
		END_IF

	30:
		Initialize := TRUE;
END_CASE
END_METHOD

END_FUNCTION_BLOCK

// ---- POUs/MAIN.TcPOU
PROGRAM MAIN
VAR
	Machine : FB_Machine := (Name := 'Machine');
END_VAR

(*All sample code provided by Beckhoff Automation LLC are for illustrative purposes only and are provided “as is” and without any warranties, express or implied. Actual implementations in applications will vary significantly. Beckhoff Automation LLC shall have no liability for, and does not waive any rights in relation to, any code samples that it provides or the use of such code samples for any purpose.*)

(*
Nain Drive: A Virtual Axis (MachineVirtualAxis) that runs a reversing sequence from 0 - 1080, with the velocity set by the Visu.

Station 1: Coupled to MachineVirtualAxis at a fixed gear ratio.

Station 2: Coupled to MachineVirtualAxis at a variable gear ratio, adjustable in the Visu.

Station 3: The Cam table master is the MachineVirtualAxis, the Virtual Cammed Axis follows the cam table. The Cammed Axis is coupled to the Virtual Cammed Axis.

Station 4: The Offset Axis is coupled to both the MachineVirtualAxis and the Virtual Offset Master Axis, and will follow commands from both of them.

Station 5: Combines 3 & 4. The Cam table master is the MachineVirtualAxis, the Virtual Cammed Axis follows the cam table. 
	The Cammed Axis is coupled to the Virtual Cammed Axis and to the Virtual Master Offset Axis.



V_Machine:
	The State Machine will begin in Aborted.
	Press the Reset button and it will progress to Idle.
	Press the Start button and it will progress to Running.
	The Machine Virtual Axis will begin its movement.
	

V_Operation:

	Notes: 
		1) The bar displays may lag behind the actual value of the axis. Use Scope View for accurate values.
		2) More details about the implementation and design choices can be found in the body of each Equipment Module (Station).
		3) While only Station 2 uses an adjustable gear ratio, it is possible to set and/or change the gear ratio of any FB_Component_BasicSlaveAxis.
			Internally the component uses MC_GearInDyn which allows for the gear ratio to be changed at any time, but does take more than 1 PLC cycle to complete.
		4) While many move types and commands (through cam tables or gear ratios) are possible to calculate and might work in a simulation, they might not work with actual hardware.
			A slave axis (whether geared or cammed) will attempt to follow the commands calculated by the NC without consideration for the physical limits of the hardware.
			Therefore, if the gear ratio is set too high then it is possible that the velocity required will cause the axis to fault.
	
		
		
	The Velocity of the Machine Virtual Axis can be changed, and the motion will run continuously from 1 to 1080.

	Station 1 
		The Fixed Axis will follow the Machine Virtual Axis at a fixed gear ratio of 0.5, therefore the value will range from 0 to 500.
 
	Station 2 
		The Variable Axis will follow the Machine Virtual Axis at an adjustable gear ratio.
		The check box for 'Change at Master 0 position' is on by default.
		The gear ratio is adjustable.
		When checked the gear ratio will change when the Machine Virtual Axis reaches 0.
		When unchecked the gear ratio will change on the next PLC scan.
		
	Station 3 
		The Virtual Cammed Axis will follow the cam table with the Machine Virtual Axis as the master axis of the table.
		The position of the master axis will be the 0 position of the table, and as the master moves the slave will follow based on the table values/calculations.
		The Cammed Axis will be geared to the Virtual Cammed Axis at the default ratio of 1:1.
		
	Station 4
		The Virtual Offset Master Axis can be moved -/+ 100 with the provided buttons.
		The Offset Axis is geared to the Machine Virtual Axis and to the Virtual Offset Master Axis, both with the default gear ratio of 1:1.
		When the Virtual Offset Master Axis is moved, the Offset Axis will apply this move to any commands received from the Machine Virtual Axis.
		This means if the Machine Virtual Axis is moving forward at 100 mm/s and the Virtual Offset Master Axis also moves forward at 100 mm/s, then the Offset Axis will move forward at 200 mm/s.
			If the Machine Virtual Axis is moving forward and the Virtual Offset Master Axis is moving in reverse at the same speed, then the Offset Axis velocity will be 0 mm/s.
	
	Station 5
		The Virtual Cammed Master Axis will follow the cam table with the Machine Virtual Axis as the master axis of the table.
		The position of the master axis will be the 0 position of the table, and as the master moves the slave will follow based on the table values/calculations.
		The Virtual Offset Master Axis can be moved -/+ 100 with the provided buttons.
		The Cammed Offset Axis will be geared to the Virtual Cammed Master Axis and to the Virtual Offset Master Axis at the default ratio of 1:1.
		This will allow the Cammed Offset Axis to follow the Cam table while also using an offset.
		
		
*)

//This is for debug only and should be removed
_AppInfo.KeepOutputsOnBP := TRUE;

//
Machine.CyclicLogic();

END_PROGRAM

// ---- VISUs/V_Operation.TcVIS
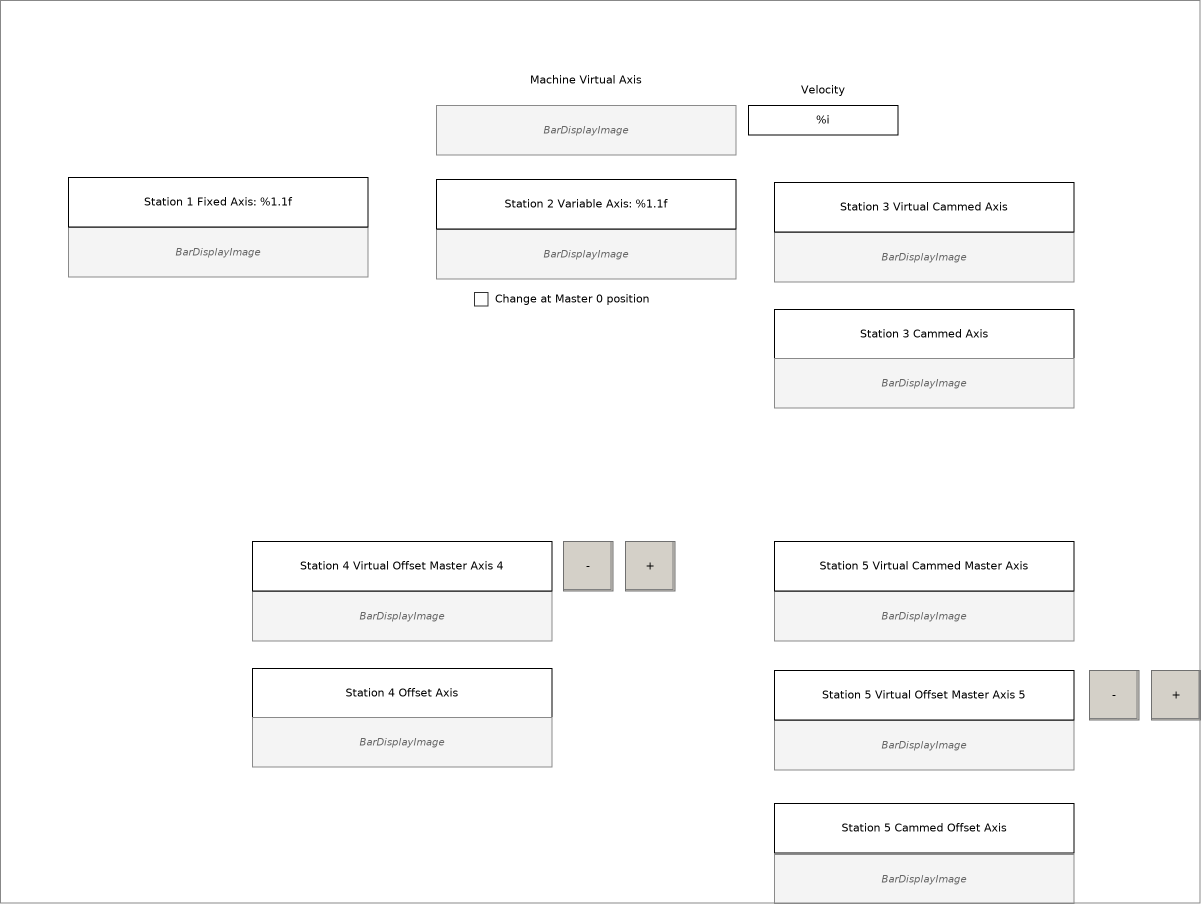
VISUALIZATION V_Operation  // 1201x904
    BarDisplayImage (436,105 300x50), value: MAIN.Machine.MainDrive.MachineVirtualAxis.AxisBase_HMI.Status.ActualPosition, style: BarDisplayImage-Gray, scale format: %.1f, scale 0..1000
    Label (436,55 300x50), "Machine Virtual Axis"
    BarDisplayImage (68,227 300x50), value: MAIN.Machine.Station1.FixedAxis.AxisBase_HMI.Status.ActualPosition, style: BarDisplayImage-Gray, scale format: %.1f, scale 0..1000
    Rectangle (68,177 300x50), "Station 1 Fixed Axis: %1.1f", text variable: MAIN.Machine.Station1.FixedAxis.BasicSlaveAxis._RatioMaster1
    BarDisplayImage (436,229 300x50), value: MAIN.Machine.Station2.VariableAxis.AxisBase_HMI.Status.ActualPosition, style: BarDisplayImage-Gray, scale format: %.1f, scale -2000..2000
    Rectangle (436,179 300x50), "Station 2 Variable Axis: %1.1f", text variable: MAIN.Machine.Station2.variableGearRatio
        OnMouseClick: write the text variable via VisuDialogs.Numpad, min -2.0, max 2.0
    BarDisplayImage (774,232 300x50), value: MAIN.Machine.Station3.VirtualCammedAxis.AxisBase_HMI.Status.ActualPosition, style: BarDisplayImage-Gray, scale format: %.1f, scale 0..100
    Rectangle (774,182 300x50), "Station 3 Virtual Cammed Axis", text variable: MAIN.Machine.Station2.VariableAxis.BasicSlaveAxis._RatioMaster1
    Rectangle (774,309 300x50), "Station 3 Cammed Axis", text variable: MAIN.Machine.Station3.CammedAxis.AxisBase_HMI.Status.ActualPosition
    BarDisplayImage (774,358 300x50), value: MAIN.Machine.Station3.CammedAxis.AxisBase_HMI.Status.ActualPosition, style: BarDisplayImage-Gray, scale format: %.1f, scale 0..150
    BarDisplayImage (252,591 300x50), value: MAIN.Machine.Station4.VirtualOffsetMasterAxis.AxisBase_HMI.Status.ActualPosition, style: BarDisplayImage-Gray, scale format: %.1f, scale 0..1000
    Rectangle (252,541 300x50), "Station 4 Virtual Offset Master Axis 4", text variable: MAIN.Machine.Station2.VariableAxis.BasicSlaveAxis._RatioMaster1
    Rectangle (252,668 300x50), "Station 4 Offset Axis", text variable: MAIN.Machine.Station3.CammedAxis.AxisBase_HMI.Status.ActualPosition
    BarDisplayImage (252,717 300x50), value: MAIN.Machine.Station4.OffsetAxis.AxisBase_HMI.Status.ActualPosition, style: BarDisplayImage-Gray, scale format: %.1f, scale 0..2000
    BarDisplayImage (774,591 300x50), value: MAIN.Machine.Station5.VirtualCammedMasterAxis.AxisBase_HMI.Status.ActualPosition, style: BarDisplayImage-Gray, scale format: %.1f, scale 0..100
    Rectangle (774,541 300x50), "Station 5 Virtual Cammed Master Axis", text variable: MAIN.Machine.Station2.VariableAxis.BasicSlaveAxis._RatioMaster1
    Rectangle (774,803 300x50), "Station 5 Cammed Offset Axis", text variable: MAIN.Machine.Station3.CammedAxis.AxisBase_HMI.Status.ActualPosition
    BarDisplayImage (774,720 300x50), value: MAIN.Machine.Station5.VirtualOffsetMasterAxis.AxisBase_HMI.Status.ActualPosition, style: BarDisplayImage-Gray, scale format: %.1f, scale 0..1000
    Rectangle (774,670 300x50), "Station 5 Virtual Offset Master Axis 5", text variable: MAIN.Machine.Station2.VariableAxis.BasicSlaveAxis._RatioMaster1
    BarDisplayImage (774,854 300x50), value: MAIN.Machine.Station5.CammedOffsetAxis.AxisBase_HMI.Status.ActualPosition, style: BarDisplayImage-Gray, scale format: %.1f, scale 0..1000
    Rectangle (748,105 150x30), "%i", text variable: MAIN.Machine.MainDrive.MachineVirtualAxis.BasicAxis._Velocity
        OnMouseClick: write the text variable via VisuDialogs.Numpad, min 0, max 100
    Checkbox (472,284 229x30), "Change at Master 0 position", variable: MAIN.Machine.Station2.sync
    Label (748,75 150x30), "Velocity"
    Button (563,541 50x50), "-"
        tap MAIN.Machine.Station4.V_OffsetREV
    Button (625,541 50x50), "+"
        tap MAIN.Machine.Station4.V_OffsetFWD
    Button (1089,670 50x50), "-"
        tap MAIN.Machine.Station5.V_OffsetREV
    Button (1151,670 50x50), "+"
        tap MAIN.Machine.Station5.V_OffsetFWD
END_VISUALIZATION

// ---- VISUs/V_Machine.TcVIS
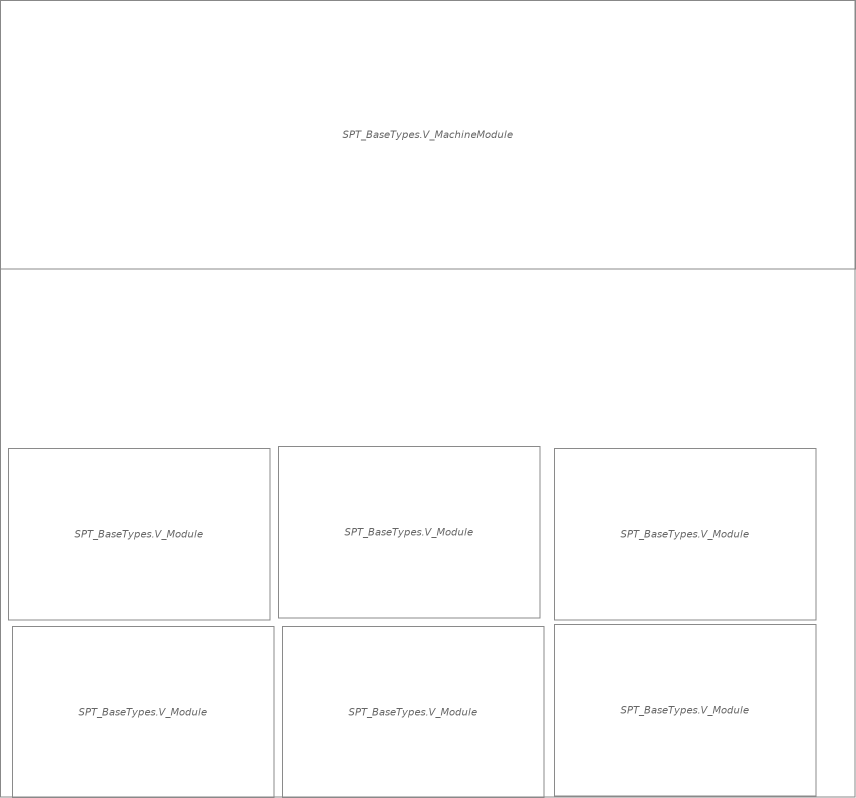
VISUALIZATION V_Machine  // 856x798
    Frame (0,0 856x269)
        shows SPT_BaseTypes.V_MachineModule(HMI := MAIN.Machine.PackMLBaseModule_HMI)
    Frame (8,448 262x172)
        shows SPT_BaseTypes.V_Module(HMI := MAIN.Machine.MainDrive.PackMLBaseModule_HMI)
    Frame (278,446 262x172)
        shows SPT_BaseTypes.V_Module(HMI := MAIN.Machine.Station1.PackMLBaseModule_HMI)
    Frame (12,626 262x172)
        shows SPT_BaseTypes.V_Module(HMI := MAIN.Machine.Station3.PackMLBaseModule_HMI)
    Frame (282,626 262x172)
        shows SPT_BaseTypes.V_Module(HMI := MAIN.Machine.Station4.PackMLBaseModule_HMI)
    Frame (554,448 262x172)
        shows SPT_BaseTypes.V_Module(HMI := MAIN.Machine.Station2.PackMLBaseModule_HMI)
    Frame (554,624 262x172)
        shows SPT_BaseTypes.V_Module(HMI := MAIN.Machine.Station5.PackMLBaseModule_HMI)
END_VISUALIZATION
